# B&R Automation Studio project hdfsjk
Automation Studio 4.10.2.37; technology packages: Acp10Arnc0 5.2.1

## Configuration Config1

CPU 4PP065.0571-P74, AutomationRuntime D4.52, Build 4.1.2, Safety 1.10, Vc V4.52.0

### Task classes (Cpu.sw)
```
Cyclic#1 (cycle 2000 us, tolerance 0 us):
  Program <- Program.prg
  ncsdcctrl <- ncsdcctrl.prg
DataObjects: Acp10sys
NcDataObjects: acp10etxen <- acp10etxen.dob, gAxis01a <- gAxis01obj.gAxis01a.dob, gAxis01i <- gAxis01obj.gAxis01i.dob, gAxis02a <- gAxis02obj.gAxis02a.dob, gAxis02i <- gAxis02obj.gAxis02i.dob
Binaries: TCData, udbdef, acp10cfg, Acp10map, iomap, arconfig, asfw, ashwac, sysconf, User, Role, ashwd
Libraries: Acp10man, Acp10par, NcGlobal, Acp10sdc, Acp10_MC, brsystem, sys_lib, runtime, AsBrStr, MotorCl, astime, fileio, powerlnk, asieccon
```

### Hardware
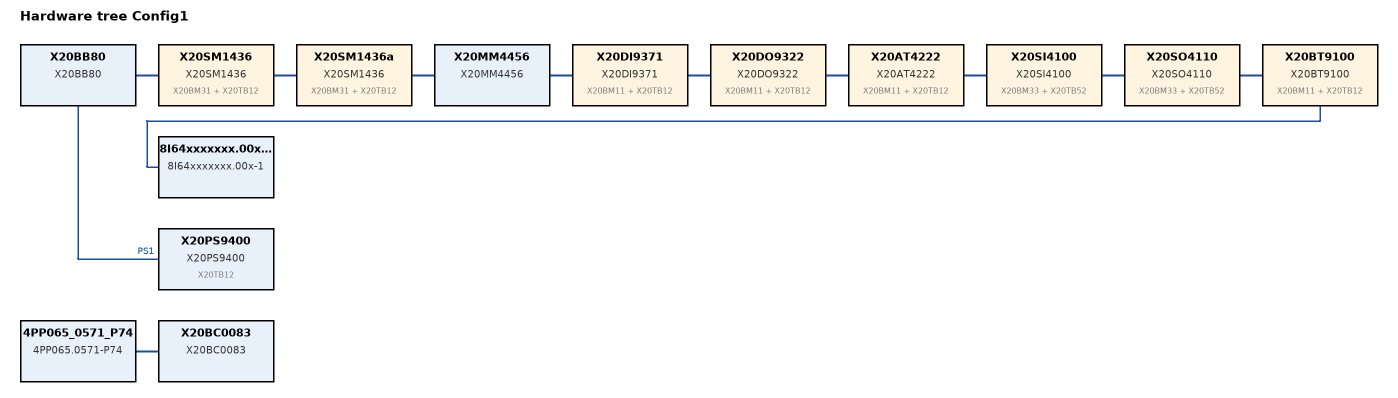
```
4PP065_0571_P74 : 4PP065.0571-P74 v1.1.2.0
  Connector IF4:
    DNAConfiguration = manual
  Connector IF5:
    ActivateDevice = 1
  ConfigurationID = hdfsjk_Config1
  Simulation = 1
  TimerDeviceType = EPLX2X
  TimerDevice = 4PP065_0571_P74.IF4
  TaskClassIdleTime = 2000
  Cyclic1Duration = 2000
  Cyclic1Tolerance = 0
  Cyclic1Output = 1
8I64xxxxxxx.00x-1 : 8I64xxxxxxx.00x-1 v2.1.2.0  [X2X1 -> X20BT9100.X2X1 [Cable Type=X2XCable, Length=10, Version=1.0.0.3]]
  FunctionModel = Standard
X20AT4222 : X20AT4222 v1.2.3.0  [SS1 -> X20TB12e.SS; SL -> X20BM11b.SL1]
X20BB80 : X20BB80 v1.0.2.0
X20BC0083 : X20BC0083 v2.9.0.0  [PLK1 -> 4PP065_0571_P74.IF4 [Cable Type=PowerlinkCable, Length=10, Version=1.0.0.3]; SL -> X20BB80.SL1]
X20BM11 : X20BM11 v1.0.0.1  [X2X1 -> X20MM4456.X2X2]
X20BM11a : X20BM11 v1.0.0.1  [X2X1 -> X20BM11.X2X2]
X20BM11b : X20BM11 v1.0.0.1  [X2X1 -> X20BM11a.X2X2]
X20BM11c : X20BM11 v1.0.0.1  [X2X1 -> X20BM33a.X2X2]
X20BM31 : X20BM31 v1.0.0.1  [X2X1 -> X20BB80.IF1]
X20BM31a : X20BM31 v1.0.0.1  [X2X1 -> X20BM31.X2X2]
X20BM33 : X20BM33 v1.1.0.0  [X2X1 -> X20BM11b.X2X2]
X20BM33a : X20BM33 v1.1.0.0  [X2X1 -> X20BM33.X2X2]
X20BT9100 : X20BT9100 v1.2.0.0  [SS1 -> X20TB12f.SS; SL -> X20BM11c.SL1]
X20DI9371 : X20DI9371 v1.0.2.0  [SS1 -> X20TB12c.SS; SL -> X20BM11.SL1]
X20DO9322 : X20DO9322 v1.0.3.0  [SS1 -> X20TB12d.SS; SL -> X20BM11a.SL1]
X20MM4456 : X20MM4456 v1.1.5.0  [X2X1 -> X20BM31a.X2X2]
X20PS9400 : X20PS9400 v1.7.0.0  [SS1 -> X20TB12.SS; PS -> X20BB80.PS1]
X20SI4100 : X20SI4100 v1.10.1.1  [SS1 -> X20TB52a.SS; SL -> X20BM33.SL1]
X20SM1436 : X20SM1436 v1.4.2.1  [SS1 -> X20TB12a.SS; SL -> X20BM31.SL1]
X20SM1436a : X20SM1436 v1.4.2.1  [SS1 -> X20TB12b.SS; SL -> X20BM31a.SL1]
X20SO4110 : X20SO4110 v1.10.1.1  [SS1 -> X20TB52b.SS; SL -> X20BM33a.SL1]
  SafeModuleID = 3
X20TB12 : X20TB12 v1.0.0.0
X20TB12a : X20TB12 v1.0.0.0
X20TB12b : X20TB12 v1.0.0.0
X20TB12c : X20TB12 v1.0.0.0
X20TB12d : X20TB12 v1.0.0.0
X20TB12e : X20TB12 v1.0.0.0
X20TB12f : X20TB12 v1.0.0.0
X20TB52a : X20TB52 v1.0.0.1
X20TB52b : X20TB52 v1.0.0.1
```

## Logical view

Binary libraries used (declarations not repeated): operator, runtime, astime, AsIecCon, Acp10man, Acp10par, NcGlobal, Acp10sdc, Acp10_MC, brsystem, sys_lib, AsBrStr

### Package Logical/Libraries - Global libraries

### Library Logical/Libraries/MotorCl (ANSIC)

#### MotorCl.fun - Exported functions and function blocks
```iecst
{REDUND_ERROR} FUNCTION_BLOCK FB_Motor (*Math model of  motor*) (*$GROUP=User,$CAT=User,$GROUPICON=User.png,$CATICON=User.png*)
	VAR_INPUT
		u : {REDUND_UNREPLICABLE} REAL;
		enable : {REDUND_UNREPLICABLE} BOOL;
	END_VAR
	VAR_OUTPUT
		w : {REDUND_UNREPLICABLE} REAL;
		phi : {REDUND_UNREPLICABLE} REAL;
	END_VAR
	VAR
		integrator : {REDUND_UNREPLICABLE} FB_Integrator;
		Tm : {REDUND_UNREPLICABLE} REAL;
		ke : {REDUND_UNREPLICABLE} REAL;
		dt : REAL;
	END_VAR
END_FUNCTION_BLOCK

{REDUND_ERROR} FUNCTION_BLOCK FB_Regulator (*PID regulator*) (*$GROUP=User,$CAT=User,$GROUPICON=User.png,$CATICON=User.png*)
	VAR_INPUT
		e : REAL;
	END_VAR
	VAR_OUTPUT
		u : REAL;
	END_VAR
	VAR
		kp : {REDUND_UNREPLICABLE} REAL;
		ki : {REDUND_UNREPLICABLE} REAL;
		integrator : {REDUND_UNREPLICABLE} FB_Integrator;
		iyOld : {REDUND_UNREPLICABLE} REAL;
		max_abs_value : {REDUND_UNREPLICABLE} REAL;
		dt : {REDUND_UNREPLICABLE} REAL;
	END_VAR
END_FUNCTION_BLOCK

{REDUND_ERROR} FUNCTION_BLOCK FB_Integrator (*Integrator*) (*$GROUP=User,$CAT=User,$GROUPICON=User.png,$CATICON=User.png*)
	VAR_INPUT
		in : {REDUND_UNREPLICABLE} REAL;
	END_VAR
	VAR_OUTPUT
		out : {REDUND_UNREPLICABLE} REAL;
	END_VAR
	VAR
		dt : {REDUND_UNREPLICABLE} REAL;
		old_err : REAL;
	END_VAR
END_FUNCTION_BLOCK

{REDUND_ERROR} {REDUND_UNREPLICABLE} FUNCTION_BLOCK FB_motor2 (*TODO: Add your comment here*) (*$GROUP=User,$CAT=User,$GROUPICON=User.png,$CATICON=User.png*)
	VAR_INPUT
		u : {REDUND_UNREPLICABLE} REAL;
		enable : {REDUND_UNREPLICABLE} BOOL;
	END_VAR
	VAR_OUTPUT
		w : {REDUND_UNREPLICABLE} REAL;
		phi : {REDUND_UNREPLICABLE} REAL;
	END_VAR
	VAR
		integrator : {REDUND_UNREPLICABLE} FB_Integrator;
		Tm : {REDUND_UNREPLICABLE} REAL;
		ke : {REDUND_UNREPLICABLE} REAL;
		dt : REAL;
	END_VAR
END_FUNCTION_BLOCK
```

#### FB_Motor.c
```c
#include <bur/plctypes.h>
#ifdef __cplusplus
	extern "C"
	{
#endif
	#include "MotorCl.h"
#ifdef __cplusplus
	};
#endif
/* Math model of  motor */
void FB_Motor(struct FB_Motor* inst)
{
	REAL variable;

	variable = inst->u/inst->ke;
	variable = variable - inst->w;
	variable = variable * inst->dt/inst->Tm;
	inst->integrator.in = variable;
	inst->integrator.dt = inst->dt;
	FB_Integrator(&inst->integrator);
	variable=inst->integrator.out;
	FB_Integrator(&inst->integrator);
	inst->w=variable;

	inst->integrator.in=inst->w * inst->dt;
	FB_Integrator(&inst->integrator);
	inst->phi+=inst->integrator.out;
	FB_Integrator(&inst->integrator);
}
```

#### FB_Regulator.c
```c
#include <bur/plctypes.h>
#ifdef __cplusplus
	extern "C"
	{
#endif
	#include "MotorCl.h"
#ifdef __cplusplus
	};
#endif
/* PID regulator */
void FB_Regulator(struct FB_Regulator* inst)
{
	REAL variable;

	variable = inst->e*inst->ki*inst->dt;
	variable += inst->iyOld;
	inst->integrator.in=variable;
	inst->integrator.dt=inst->dt;
	FB_Integrator(&inst->integrator);

	if(inst->e*inst->kp>inst->max_abs_value)
	{

		variable=inst->integrator.out+inst->max_abs_value;
			FB_Integrator(&inst->integrator);
	}
	if(inst->e*inst->kp<inst->max_abs_value)
	{
		variable=inst->integrator.out+inst->e*inst->kp;
			FB_Integrator(&inst->integrator);
	}
	if(variable>inst->max_abs_value)
	{
		inst->u=inst->max_abs_value;
		inst->iyOld=variable-inst->max_abs_value;
	}
	else
	{
		inst->u=variable;
		inst->iyOld=0;
	}
}
```

#### FB_Integrator.c
```c
#include <bur/plctypes.h>
#ifdef __cplusplus
	extern "C"
	{
#endif
	#include "MotorCl.h"
#ifdef __cplusplus
	};
#endif
/* Integrator */
void FB_Integrator(struct FB_Integrator* inst)
{
	inst-> out = inst->old_err + (inst->in)* inst->dt;
	inst->old_err= inst->out;

}
```

#### FB_motor2.c
```c
#include <bur/plctypes.h>
#ifdef __cplusplus
	extern "C"
	{
#endif
	#include "MotorCl.h"
#ifdef __cplusplus
	};
#endif
/* TODO: Add your comment here */
void FB_motor2(struct FB_motor2* inst)

	{
		REAL variable;

		variable = inst->u/inst->ke;
		variable = variable - inst->w;
		variable = variable * inst->dt/inst->Tm;
		inst->integrator.in = variable;
		inst->integrator.dt = inst->dt;
		FB_Integrator(&inst->integrator);
		variable=inst->integrator.out;
		FB_Integrator(&inst->integrator);
		inst->w=variable;

		inst->integrator.in=inst->w * inst->dt;
		FB_Integrator(&inst->integrator);
		inst->phi+=inst->integrator.out;
		FB_Integrator(&inst->integrator);
	}
```

### Program Logical/Program (ANSIC)

#### Variables.var
```iecst
VAR
	fb_regulator : FB_Regulator;
	fb_motor : FB_Motor;
	Speed : REAL;
	enable : BOOL;
	t : REAL;
	fb_motor2 : FB_motor2;
END_VAR
```

#### Main.c
```c
#include <bur/plctypes.h>

#ifdef _DEFAULT_INCLUDES
	#include <AsDefault.h>
#endif

void _INIT ProgramInit(void)
{
	REAL t;

	Speed=200;
	t=0;

	fb_regulator.dt =0.002;
	fb_regulator.e=10;
	fb_regulator.ki=0.16;
	fb_regulator.kp=0.0064;
	fb_regulator.max_abs_value=300;

	fb_motor.dt=0.002;
	fb_motor.Tm=0.04;
	fb_motor.ke = (fb_regulator.ki*3*fb_regulator.dt);

	fb_motor2.dt=0.002;
	fb_motor2.Tm=0.04;
	fb_motor2.ke = (fb_regulator.ki*3*fb_regulator.dt);
}

void _CYCLIC ProgramCyclic(void)
{

	if (enable == 1)
	{
		Speed = 200;
	}
	else
	{
		Speed = 0;
	}
	t=t+0.001;
	fb_regulator.e=Speed-fb_motor.w;
	FB_Regulator(&fb_regulator);
	fb_motor.u=fb_regulator.u;
	FB_Motor(&fb_motor);
	fb_motor2.u = Speed-fb_motor2.w;
	FB_motor2(&fb_motor2);

	if((t>=5)&&(t<10))
	{
		enable = 1;
	}
	if ((t>=10)&&(t<15))
	{
		enable = 0;
	}
	if (t>=15)
	{
		enable = 1;
		t = 0;
	}
}

void _EXIT ProgramExit(void)
{

}
```

Listed in the project but not available here: Logical/Libraries/MotorCl/Types.typ, Logical/Libraries/MotorCl/Constants.var, Logical/ncsdcctrl, Logical/acp10etxen, Logical/gAxis01obj, Logical/gAxis02obj, Logical/Global.typ, Logical/Global.var
